// SIMATIC S7-200 project (STEP 7-Micro/WIN), CPU 224XP REL 02.01

SUBROUTINE_BLOCK SCALE:SBR0
TITLE=COMENTARIOS DE LA SUBRUTINA
VAR_INPUT
X2_VMAX:REAL;	// LD0 
X1_VMIN:REAL;	// LD4 
Y2_VMAX:REAL;	// LD8 
Y1_VMIN:REAL;	// LD12 
IN_VX:REAL;	// LD16 
END_VAR
VAR_OUTPUT
OUT_Y:REAL;	// LD20 
END_VAR
VAR
Y2_Y1:REAL;	// LD24 
X2_X1:REAL;	// LD28 
M:REAL;	// LD32 
MX2:REAL;	// LD36 
N:REAL;	// LD40 
END_VAR
BEGIN
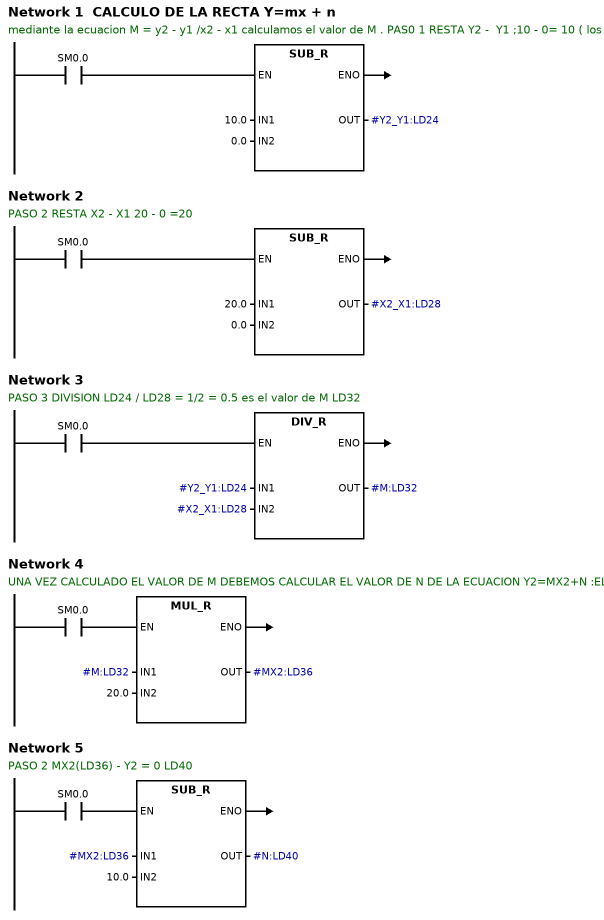
Network 1 // CALCULO DE LA RECTA Y=mx + n 
// mediante la ecuacion M = y2 - y1 /x2 - x1 calculamos el valor de M . PAS0 1 RESTA Y2 -  Y1 ;10 - 0= 10 ( los valores de y2,y1,x2,x1 son referencias para poder calcular el valor de M )
LD     SM0.0
MOVR   10.0, #Y2_Y1:LD24
-R     0.0, #Y2_Y1:LD24
Network 2
// PASO 2 RESTA X2 - X1 20 - 0 =20
LD     SM0.0
MOVR   20.0, #X2_X1:LD28
-R     0.0, #X2_X1:LD28
Network 3
// PASO 3 DIVISION LD24 / LD28 = 1/2 = 0.5 es el valor de M LD32
LD     SM0.0
MOVR   #Y2_Y1:LD24, #M:LD32
/R     #X2_X1:LD28, #M:LD32
Network 4
// UNA VEZ CALCULADO EL VALOR DE M DEBEMOS CALCULAR EL VALOR DE N DE LA ECUACION Y2=MX2+N :EL VALOR  DESPEJANDO SERIA N=MX2 -Y2; 0.5*20 -10=0 PASO 1 M + X2 LD36
// (network saved uncompiled; LAD cells follow)
// row 0: c0 -| |- SM0.0  c1 [MUL_R EN:=power@row0, IN1:=#M:LD32, IN2:=20.0, ENO=>power, OUT=>#MX2:LD36]  c2 ->
// row 1: c1 [box]
Network 5
// PASO 2 MX2(LD36) - Y2 = 0 LD40
// (network saved uncompiled; LAD cells follow)
// row 0: c0 -| |- SM0.0  c1 [SUB_R EN:=power@row0, IN1:=#MX2:LD36, IN2:=10.0, ENO=>power, OUT=>#N:LD40]  c2 ->
// row 1: c1 [box]
Network 6
// EL SIGUIENTE PASO NOS PERMITIRA AVERIGUAR EL VALOR DE Y RESPECTO A X ,COMO YA TENEMOS M Y N SIMPLEMENTE TENEMOS QUE APLICAR LA ECUACION DE LA RECTA
END_SUBROUTINE_BLOCK
